SUBAPPLICATION VirendraTests (* Subapplication Type *)
  (* Standard: 61499-2 *)
  (* Version 1.0, 2025-05-16, az *)
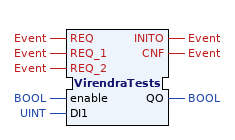
  EVENT_INPUT
    REQ; (* Normal Execution Request *)
    REQ_1;
    REQ_2;
  END_EVENT
  EVENT_OUTPUT
    INITO; (* Initialization Confirm *)
    CNF; (* Execution Confirmation *)
  END_EVENT
  VAR_INPUT
    enable : BOOL; (* Input event qualifier *)
    DI1 : UINT;
  END_VAR
  VAR_OUTPUT
    QO : BOOL; (* Output event qualifier *)
  END_VAR
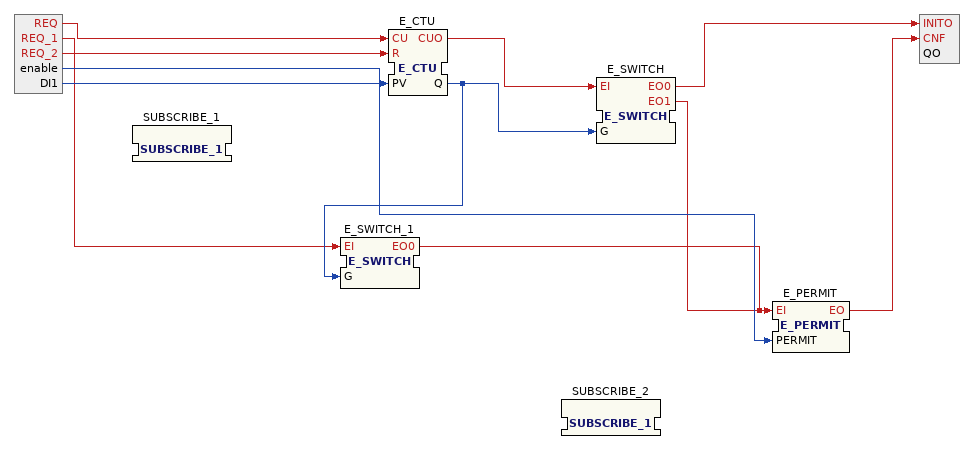
  FBS
    E_PERMIT : E_PERMIT;
    E_CTU : E_CTU;
    E_SWITCH : E_SWITCH;
    E_SWITCH_1 : E_SWITCH;
    SUBSCRIBE_1 : SUBSCRIBE_1;
    SUBSCRIBE_2 : SUBSCRIBE_1;
  END_FBS
  EVENT_CONNECTIONS
    REQ TO E_CTU.CU;
    E_CTU.CUO TO E_SWITCH.EI;
    E_SWITCH.EO0 TO INITO;
    E_SWITCH.EO1 TO E_PERMIT.EI;
    E_PERMIT.EO TO CNF;
    REQ_1 TO E_SWITCH_1.EI;
    REQ_2 TO E_CTU.R;
    E_SWITCH_1.EO0 TO E_PERMIT.EI;
  END_CONNECTIONS
  DATA_CONNECTIONS
    DI1 TO E_CTU.PV;
    enable TO E_PERMIT.PERMIT;
    E_CTU.Q TO E_SWITCH.G;
    E_CTU.Q TO E_SWITCH_1.G;
  END_CONNECTIONS
END_SUBAPPLICATION
